(* PLC project liner_cyclic.project, CODESYS CODESYS V3.5 SP17 Patch 3 *)
(* stored: creationDateTime 1970-01-01T00:00:00, modificationDateTime 1970-01-01T00:00:00 *)

FUNCTION_BLOCK qqq
  VAR
    a : INT;
    b : INT;
  END_VAR

            a := b + 6;
          
END_FUNCTION_BLOCK
